Omron CX-Programmer project NewProject (CX-Programmer 9.61)

# PLC NewPLC1: CP1L M

## Global symbols (name address type ; comment)
Block FunctionBlock1
TIM FunctionBlock1
block FunctionBlock1

## Program NewProgram1 (cyclic task 0)
Local symbols
C1_dir 100.00 BOOL
C1_esq 100.01 BOOL
C2_des 100.02 BOOL
C2_sub 100.03 BOOL
C3_des 100.05 BOOL
C3_sub 100.04 BOOL
C4_ 100.06 BOOL
EN BOOL
LedGreen 101.00 BOOL
LedRed 100.07 BOOL
LedYellow 101.01 BOOL
P_ON BOOL
S10_ 0.07 BOOL
S14_ 0.09 BOOL
S15_ 0.10 BOOL
S5_ 0.02 BOOL
S7_ 0.04 BOOL
S8_ 0.05 BOOL
S9_ 0.06 BOOL
Start 0.00 BOOL
Stop 0.01 BOOL
ctime 201.00 BOOL
ctimefim BOOL
s13_ 0.08 BOOL

### Section Section1

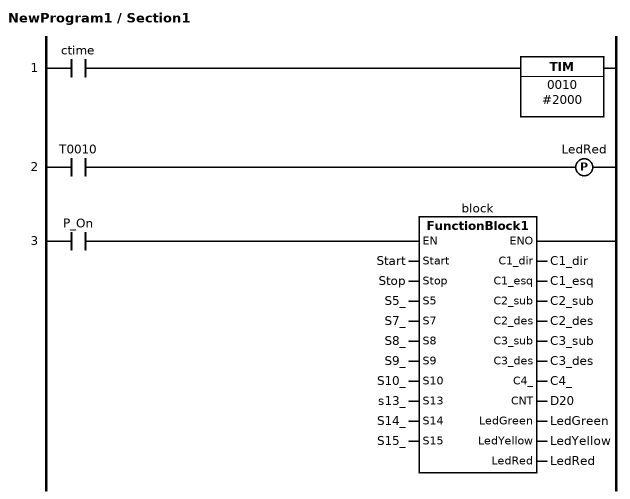
; rung 1
LD ctime
TIM 0010 #2000
; rung 2
LD T0010
DIFU(013) LedRed
; rung 3
LD P_On
CALL block : FunctionBlock1 (Start := Start, Stop := Stop, S5 := S5_, S7 := S7_, S8 := S8_, S9 := S9_, S10 := S10_, S13 := s13_, S14 := S14_, S15 := S15_, C1_dir => C1_dir, C1_esq => C1_esq, C2_sub => C2_sub, C2_des => C2_des, C3_sub => C3_sub, C3_des => C3_des, C4_ => C4_, CNT => D20, LedGreen => LedGreen, LedYellow => LedYellow, LedRed => LedRed)

### Section END
; rung 0
END(001)

## Function block FunctionBlock1
VAR_INPUT
  Start : BOOL;
  Stop : BOOL;
  S5 : BOOL := TRUE;
  S7 : BOOL := TRUE;
  S8 : BOOL;
  S9 : BOOL := TRUE;
  S10 : BOOL;
  S13 : BOOL;
  S14 : BOOL;
  S15 : BOOL;
END_VAR
VAR_OUTPUT
  C1_dir : BOOL;
  C1_esq : BOOL;
  C2_sub : BOOL;
  C2_des : BOOL;
  C3_sub : BOOL;
  C3_des : BOOL;
  C4_ : BOOL;
  CNT : INT;
  LedGreen : BOOL;
  LedYellow : BOOL;
  LedRed : BOOL;
  ctime : BOOL;
END_VAR
VAR
  EstadoAtivo : INT;
END_VAR
IF(EstadoAtivo=0 )OR( EstadoAtivo=2 AND S7=FALSE) OR (EstadoAtivo=6 AND S7= FALSE) OR( EstadoAtivo=14 AND S5=FALSE) THEN
	EstadoAtivo:=0;
	C1_dir:= FALSE;
	C1_esq:= FALSE;
	C2_sub:= FALSE;
	C2_des:= FALSE;
	C3_des:= FALSE;
	C3_sub:= FALSE;
	C4_:= FALSE;
	LedGreen:= FALSE;
	LedRed:= FALSE;
	LedYellow:= FALSE;
	CNT:= 0;

END_IF;

IF(EstadoAtivo=0 AND Start=TRUE AND Stop=FALSE AND S7=TRUE AND S15=TRUE)THEN
	
	EstadoAtivo:=1;
	C1_dir:= FALSE;
	C1_esq:= FALSE;
	C2_sub:= FALSE;
	C2_des:= TRUE;
	C3_des:= FALSE;
	C3_sub:= FALSE;
	C4_:= FALSE;
	LedGreen:= FALSE;
	LedRed:= FALSE;
	LedYellow:= FALSE;
	
END_IF;
(*estado2*)
IF(EstadoAtivo= 1 OR EstadoAtivo=3 OR EstadoAtivo=11)AND( S8=TRUE AND Stop= TRUE)THEN
	EstadoAtivo:=2;
	C1_dir:= FALSE;
	C1_esq:= FALSE;
	C2_sub:= TRUE;
	C2_des:= FALSE;
	C3_des:= FALSE;
	C3_sub:= FALSE;
	C4_:= FALSE;
	LedGreen:= FALSE;
	LedRed:= FALSE;
	LedYellow:= FALSE;
END_IF;
(*estado*)
IF(EstadoAtivo=1 AND S8=FALSE AND S5= TRUE AND Stop=FALSE)THEN
	EstadoAtivo:=3;
	C1_dir:= TRUE;
	C1_esq:= FALSE;
	C2_sub:= FALSE;
	C2_des:= FALSE;
	C3_des:= FALSE;
	C3_sub:= FALSE;
	C4_:= FALSE;
	LedGreen:= FALSE;
	LedRed:= FALSE;
	LedYellow:= FALSE;
END_IF;
(*estado 4*)
IF(EstadoAtivo=3 AND S13=TRUE AND S9= TRUE AND Stop=FALSE)THEN
	EstadoAtivo:=4;
	C1_dir:= FALSE;
	C1_esq:= FALSE;
	C2_sub:= FALSE;
	C2_des:= FALSE;
	C3_des:= TRUE;
	C3_sub:= FALSE;
	C4_:= FALSE;
	LedGreen:= FALSE;
	LedRed:= FALSE;
	LedYellow:= FALSE;
END_IF;
(*estado5*)
IF(((EstadoAtivo=4 OR EstadoAtivo=7 OR EstadoAtivo=10)) AND S10=TRUE AND Stop=TRUE) THEN
	EstadoAtivo:=5;
	C1_dir:= FALSE;
	C1_esq:= FALSE;
	C2_sub:= FALSE;
	C2_des:= FALSE;
	C3_des:= FALSE;
	C3_sub:= TRUE;
	C4_:= FALSE;
	LedGreen:= FALSE;
	LedRed:= FALSE;
	LedYellow:= FALSE;
END_IF;
(*estado6*)
IF(EstadoAtivo=5 AND S9=FALSE AND S8=TRUE)THEN
	EstadoAtivo:=5;
	C1_dir:= FALSE;
	C1_esq:= FALSE;
	C2_sub:= FALSE;
	C2_des:= TRUE;
	C3_des:= FALSE;
	C3_sub:= FALSE;
	C4_:= FALSE;
	LedGreen:= FALSE;
	LedRed:= FALSE;
	LedYellow:= FALSE;
END_IF;
(*estado7*)
IF(EstadoAtivo=4 AND S10=FALSE AND Stop=FALSE)THEN
	EstadoAtivo:=7;
	C1_dir:= FALSE;
	C1_esq:= FALSE;
	C2_sub:= FALSE;
	C2_des:= FALSE;
	C3_des:= FALSE;
	C3_sub:= FALSE;
	C4_:= TRUE;
	LedGreen:= FALSE;
	LedRed:= FALSE;
	LedYellow:= FALSE;
END_IF;
(*estado8*)
IF(EstadoAtivo=7 AND S13=FALSE AND Stop=FALSE)THEN
	EstadoAtivo:=8;
	C1_dir:= FALSE;
	C1_esq:= FALSE;
	C2_sub:= FALSE;
	C2_des:= FALSE;
	C3_des:= FALSE;
	C3_sub:= FALSE;
	C4_:= FALSE;
	LedGreen:= FALSE;
	LedRed:= FALSE;
	LedYellow:= FALSE;
END_IF;
(*estado9*)
IF(EstadoAtivo=8 AND S14=TRUE AND Stop=FALSE)THEN
	EstadoAtivo:=9;
	C1_dir:= FALSE;
	C1_esq:= FALSE;
	C2_sub:= FALSE;
	C2_des:= FALSE;
	C3_des:= FALSE;
	C3_sub:= FALSE;
	C4_:= FALSE;
	LedGreen:= FALSE;
	LedRed:= FALSE;
	CNT:=CNT+1;
	LedYellow:= FALSE;
END_IF;
(*estado10*)
IF(EstadoAtivo=7 AND S13=FALSE AND Stop=FALSE)THEN
	EstadoAtivo:=10;
	C1_dir:= FALSE;
	C1_esq:= FALSE;
	C2_sub:= FALSE;
	C2_des:= FALSE;
	C3_des:=FALSE;
	C3_sub:= FALSE;
	C4_:= FALSE;
	LedGreen:= FALSE;
	LedRed:= FALSE;
	LedYellow:= FALSE;
END_IF;
(*estado11*)
IF(EstadoAtivo=10 AND S10=TRUE AND Stop=FALSE)THEN
	EstadoAtivo:=11;
	C1_dir:= FALSE;
	C1_esq:= FALSE;
	C2_sub:= FALSE;
	C2_des:= FALSE;
	C3_des:= FALSE;
	C3_sub:= TRUE;
	C4_:= FALSE;
	LedGreen:= FALSE;
	LedRed:= FALSE;
	LedYellow:= FALSE;
END_IF;
(*estado12*)
IF(EstadoAtivo=11 AND S9=FALSE AND S8=TRUE AND Stop=FALSE)THEN
	EstadoAtivo:=12;
	C1_dir:= FALSE;
	C1_esq:= FALSE;
	C2_sub:= TRUE;
	C2_des:= FALSE;
	C3_des:= FALSE;
	C3_sub:= FALSE;
	C4_:= FALSE;
	LedGreen:= FALSE;
	LedRed:= FALSE;
	LedYellow:= FALSE;
END_IF;
(*estado13*)
IF(EstadoAtivo=12 AND S7=FALSE AND Stop=FALSE)THEN
	EstadoAtivo:=13;
	C1_dir:= FALSE;
	C1_esq:= TRUE;
	C2_sub:= FALSE;
	C2_des:= FALSE;
	C3_des:= FALSE;
	C3_sub:= FALSE;
	C4_:= FALSE;
	LedGreen:= FALSE;
	LedRed:= FALSE;
	LedYellow:= FALSE;
END_IF;
(*estado14*)
IF(EstadoAtivo=12 AND Stop=TRUE)THEN
	EstadoAtivo:=14;
	C1_dir:= FALSE;
	C1_esq:= TRUE;
	C2_sub:= FALSE;
	C2_des:= FALSE;
	C3_des:= FALSE;
	C3_sub:= FALSE;
	C4_:= FALSE;
	LedGreen:= FALSE;
	LedRed:= FALSE;
	LedYellow:= FALSE;
END_IF;
(*estado15*)
IF(EstadoAtivo=9 AND EstadoAtivo=13 AND S14=FALSE AND S5 = FALSE AND Stop=FALSE)THEN
	EstadoAtivo:=15;
	C1_dir:= FALSE;
	C1_esq:= FALSE;
	C2_sub:= FALSE;
	C2_des:= FALSE;
	C3_des:= FALSE;
	C3_sub:= FALSE;
	C4_:= FALSE;
	LedGreen:= FALSE;
	LedRed:= FALSE;
	LedYellow:= FALSE;
END_IF;
(*estado16*)
IF(EstadoAtivo=15 AND Stop=FALSE AND CNT<8)THEN
	EstadoAtivo:=16;
	C1_dir:= FALSE;
	C1_esq:= FALSE;
	C2_sub:= FALSE;
	C2_des:= FALSE;
	C3_des:= FALSE;
	C3_sub:= FALSE;
	C4_:= FALSE;
	LedGreen:= TRUE;
	LedRed:= FALSE;
	LedYellow:= FALSE;
END_IF;
(*estado17*)
IF(EstadoAtivo=15 AND Stop=FALSE AND CNT=8)THEN
	EstadoAtivo:=17;
	C1_dir:= FALSE;
	C1_esq:= FALSE;
	C2_sub:= FALSE;
	C2_des:= FALSE;
	C3_des:= FALSE;
	C3_sub:= FALSE;
	C4_:= FALSE;
	LedGreen:= FALSE;
	LedRed:= FALSE;
	LedYellow:=TRUE;
END_IF;
(*estado18*)
IF(EstadoAtivo=15 AND Stop=FALSE AND CNT=10)THEN
	EstadoAtivo:=18;
	C1_dir:= FALSE;
	C1_esq:= FALSE;
	C2_sub:= FALSE;
	C2_des:= FALSE;
	C3_des:= FALSE;
	C3_sub:= FALSE;
	C4_:= FALSE;
	LedGreen:= FALSE;
	LedRed:= TRUE;
	ctime:= TRUE;
	LedYellow:=FALSE;
	CNT:= 0;
END_IF;